// SIMATIC S7-200 project (STEP 7-Micro/WIN), CPU 221 REL 01.10

SYMBOL_TABLE USER1
Start_button     I0.0     // TO START THE OUTPUT 1 AND 2
Stop_button      I0.1     // TO STOP THE OUTPUT 1
Limit_switch     I0.2     // TO STOP THE OUTPUT 2
Output_1         Q0.0
Output_2         Q0.1
Red_indicator    Q0.2     // INDICATES LIMIT SWITCH TURNED ON
END_SYMBOL_TABLE

ORGANIZATION_BLOCK MAIN:OB1
TITLE=PROGRAM COMMENTS
BEGIN
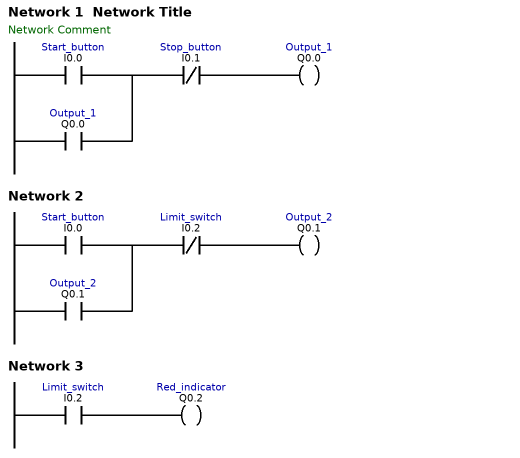
Network 1 // Network Title
// Network Comment
LD     Start_button:I0.0
O      Output_1:Q0.0
AN     Stop_button:I0.1
=      Output_1:Q0.0
Network 2
LD     Start_button:I0.0
O      Output_2:Q0.1
AN     Limit_switch:I0.2
=      Output_2:Q0.1
Network 3
LD     Limit_switch:I0.2
=      Red_indicator:Q0.2
END_ORGANIZATION_BLOCK
